PROGRAM MAIN_oo
VAR
	
	// network interface/simulator function blocks
	netiMeshCal				:FB_3eTI_iMesh_Cal;
	netiMeshTESIM			:FB_3eTI_iMesh_TESIM;
	netiMeshTestSignals		:FB_3eTI_TestSignals;
	netiMeshGasSensor		:FB_3eTI_iMesh_GasSensor;
	netiMeshLFSR			:FB_3eTI_iMesh_LFSR;
	
	netPCCal				:FB_PC_OneLink_Cal;
	netPCTESIM				:FB_PC_OneLink_TESIM;
	netPCTestSignals		:FB_PC_OneLink_TestSignals;
	netPCGasSensor			:FB_PC_OneLink_GasSensor;
	netPC_LFSR				:FB_PC_LFSR;
	
	// yokogawa signals
	netYokoTestSignals		:FB_Yokogawa_TestSignals;
	netYokoLFSR				:FB_Yokogawa_LFSR;
	netYokoGasSensor		:FB_Yokogawa_GasSensor;

	netNoNet				:FB_NoNet;
	
END_VAR



CASE NET_TYPE OF 
	100:
	netiMeshCal();
	101:
	netiMeshTESIM();
	102:
	netiMeshTestSignals();
	103:
	netiMeshGasSensor();
	110:
	netiMeshLFSR();
	
	200:
	netPCCal();
	201:
	netPCTESIM();
	202:
	netPCTestSignals();
	203:
	netPCGasSensor();	
	210:
	netPC_LFSR();
	
	300:
	301:
	302:
	netYokoTestSignals();
	303:
	netYokoGasSensor();
	310:
	netYokoLFSR();
	
	
ELSE
	netnoNet();
	
END_CASE

END_PROGRAM

(* stored: Version 1.1.0.1, ProductVersion 3.1.4020.12
   POU MAIN_oo: Id {dd06f3b9-f114-454f-820d-85f29a3eb792}, SpecialFunc None *)
